Fanuc TP program (LS listing): PRT07POUNCE.LS

/PROG  PRT07POUNCE
/ATTR
OWNER		= MNEDITOR;
COMMENT		= "POUNCE Core 311";
PROG_SIZE	= 1101;
CREATE		= DATE 20-06-20  TIME 05:48:26;
MODIFIED	= DATE 20-06-20  TIME 05:48:26;
FILE_NAME	= PRT07POU;
VERSION		= 0;
LINE_COUNT	= 26;
MEMORY_SIZE	= 1369;
PROTECT		= READ_WRITE;
STORAGE		= SHADOW;
TCD:  STACK_SIZE	= 0,
      TASK_PRIORITY	= 50,
      TIME_SLICE	= 0,
      BUSY_LAMP_OFF	= 0,
      ABORT_REQUEST	= 0,
      PAUSE_REQUEST	= 0;
DEFAULT_GROUP	= 1,*,*,*,*;
CONTROL_CODE	= 00000000 00000000;
/APPL
  HANDLING : TRUE ;
/MN
   1:  !******************************** ;
   2:  ! PATH - pounce core pick ;
   3:  !*    core (moving) end ;
   4:  !******************************** ;
   5:  !PROGRAM : PRT02POUNCE ;
   6:  !ASSEMBLY: XXXXXX ;
   7:  !ROBOT ID: F196839 ;
   8:  !******************************** ;
   9:  !MOVE TO POUNCE - PATH SEGMENT ;
  10:   ;
  11:  SET SEGMENT(1) ;
  12:  !SET SEGMENT(1), Home to Pounce ;
  13:   ;
  14:  !Set ATI Tool and World UFrame ;
  15:  UTOOL_NUM=7 ;
  16:  UFRAME_NUM=0 ;
  17:  PAYLOAD[6] ;
  18:   ;
  19:  !AT POUNCE ;
  20:J P[1:At Pounce] 70% CNT100    ;
  21:   ;
  22:  Set MH Tool(7) ;
  23:  Release Part(5) ;
  24:   ;
  25:  MESSAGE[WAITING AT POUNCE] ;
  26:  AT PICK POUNCE    ;
/POS
P[1:"At Pounce"]{
   GP1:
	UF : 0, UT : 7,		CONFIG : 'N U T, 0, 0, 0',
	X =  1180.818  mm,	Y =  2674.389  mm,	Z =   539.175  mm,
	W =  -174.091 deg,	P =    57.925 deg,	R =     1.541 deg
};
/END
